FUNCTION_BLOCK VECTOR_ABS (* Vector module *)
  (* Standard: 61499-2 *)
  (* Version 1.0, 02-05-12, GASR, Universidade do Estado de Santa Catarina *)
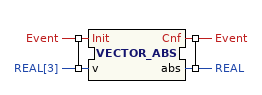
  EVENT_INPUT
    Init WITH v;
  END_EVENT
  EVENT_OUTPUT
    Cnf WITH abs;
  END_EVENT
  VAR_INPUT
    v : ARRAY [0..2] OF REAL;
  END_VAR
  VAR_OUTPUT
    abs : REAL;
  END_VAR
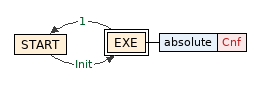
  EC_STATES
    EXE : absolute -> Cnf;
    START;
  END_STATES
  EC_TRANSITIONS
    START TO EXE := Init;
    EXE TO START := 1;
  END_TRANSITIONS
  ALGORITHM absolute IN Lua:
 abs = ( ( v[ 1 ]^2 ) + ( v[ 2 ]^2 ) + ( v[ 3 ]^2 ) )^0.5
  END_ALGORITHM
END_FUNCTION_BLOCK
